(* PLC project v0.6.02_RefactorGateAndTest.project, CODESYS CODESYS V3.5 SP19 Patch 1 *)
(* stored: creationDateTime 2026-08-14T10:10:49.355835, modificationDateTime 2026-08-14T10:10:49.355835 *)

(* ═══════════════════════════════════════════════════════════════ 🛡️ ST_Safety_Emergency_Diag — Diagnostic et erreurs de la chaîne AU ─────────────────────────────────────────────────────────────── 📄 Produit par FB_Safety_EmergencyManagement (sortie Diag). Consommé par PRG_SUPERVISION_CFC et GVL_Troubleshooting. 🎯 Champs lecture seule — producteur unique = FB composite. ═══════════════════════════════════════════════════════════════ 📄 Docs : DOC/AF/AF_Partie-01_Analyse_Fonctionnelle_v2.0.md §8.2 DOC/AF/AF_Partie-03_Contrats_Composants_v2.1.md *)
TYPE ST_Safety_Emergency_Diag : STRUCT
  Error : BOOL;  (* 🔴 Synthèse : (ErrorId <> 0) *)
  ErrorId : WORD;  (* ❌ bit0 = RedundancyTestFailed (auto-test A/B), bit1 = EmergencyArmingFailed (timeout confirm contacteur) *)
  RedundancyTestFailed : BOOL;  (* 🔴 Canal A ou B resté collé/shunté détecté à l'auto-test — Reset requis (cause disparue) *)
  ArmFailed : BOOL;  (* 🔴 Impulsion envoyée mais contacteur puissance non confirmé sous 2 s — Reset + contacteur engagé requis *)
  LockoutActive : BOOL;  (* ⏳ Verrouillage temporel de 5 s entre tentatives de réarmement échouées *)
END_STRUCT;
END_TYPE

(* ═══════════════════════════════════════════════════════════════ ⚙️ ST_Safety_Emergency_InternalCmd — Structure de commande interne ─────────────────────────────────────────────────────────────── 📄 Transporte les ordres logiques entre le bloc de décision et le bloc de sortie de la boucle d'urgence. 🔒 Polarité maintien : TRUE = voie maintenue saine, FALSE = coupure demandée (conforme règle C1 — polarité explicite). ═══════════════════════════════════════════════════════════════ 📄 Docs : DOC/AF/AF_Partie-01_Analyse_Fonctionnelle_v2.0.md *)
TYPE ST_Safety_Emergency_InternalCmd : STRUCT
  MaintainA_Cmd : BOOL;  (* Ordre maintien canal A (TRUE = voie maintenue, FALSE = coupure demandée) *)
  MaintainB_Cmd : BOOL;  (* Ordre maintien canal B (TRUE = voie maintenue, FALSE = coupure demandée) *)
  ArmPulse_Cmd : BOOL;  (* Ordre impulsion de réarmement (TRUE = bobine réarmement activée) *)
END_STRUCT;
END_TYPE

(* ═══════════════════════════════════════════════════════════════ 🚦 ST_Safety_Emergency_State — État public de la chaîne d'arrêt d'urgence ─────────────────────────────────────────────────────────────── 📄 Produit par FB_Safety_EmergencyManagement (sortie State). Consommé par PRG_SUPERVISION_CFC → GVL_IHM.Modes.State pour IHM, et par GVL_Troubleshooting pour diagnostic. 🎯 Champs lecture seule — aucun lecteur n'est autorisé à l'écrire. ═══════════════════════════════════════════════════════════════ 📄 Docs : DOC/AF/AF_Partie-01_Analyse_Fonctionnelle_v2.0.md §8.2 DOC/AF/AF_Partie-03_Contrats_Composants_v2.1.md *)
TYPE ST_Safety_Emergency_State : STRUCT
  ChainOk : BOOL;  (* 🔗 Boucle AU fermée (EmergencyChainClosed_DI = TRUE) *)
  ContactorOk : BOOL;  (* 🔌 Contacteur puissance confirmé engagé (PowerContactorEngaged_DI = TRUE) *)
  Step : INT;  (* 🔢 Étape séquence armement : 0=IDLE, 1=TestA, 2=RestoreA, 3=TestB, 4=RestoreB, 5=Pulse, 6=Confirm *)
  Armable : BOOL;  (* 🟢 Réarmement possible maintenant : chain OK, step=0, pas de lockout, pas de redondance échouée, pas de contacteur déjà engagé *)
  ArmingBusy : BOOL;  (* ⏳ Séquence armement OU lockout en cours (nouvelle demande ignorée) *)
END_STRUCT;
END_TYPE

(* ═══════════════════════════════════════════════════════════════ 🔒 FB_Safety_EmergencyManagementOutput — Projection Physique Fail-Safe ─────────────────────────────────────────────────────────────── 🎯 Rôle : Enable gate + copie consignes logiques vers sorties physiques 🔒 Polarité : MaintainA/B_RQ en maintien (TRUE = voie saine) 📄 Docs : DOC/AF/AF_Partie-01_Analyse_Fonctionnelle/FB_Safety_EmergencyManagement_v1.1.md DOC/AF/AF_Partie-01_Analyse_Fonctionnelle_v2.0.md DOC/AF/AF_Partie-03_Contrats_Composants_v2.1.md *)
FUNCTION_BLOCK FB_Safety_EmergencyManagementOutput
  VAR_INPUT
    Enable : BOOL;  (* Active le pilote (FALSE = toutes sorties à FALSE) *)
    Cmd : ST_Safety_Emergency_InternalCmd;  (* Ordres logiques reçus du bloc logique *)
    ChainOk : BOOL;  (* Miroir EmergencyChainClosed (pour bus State) *)
    ContactorOk : BOOL;  (* Miroir PowerContactorEngaged (pour bus State) *)
    ArmingStep : INT;  (* Miroir ArmingSeqStep (pour bus State) *)
    Armable : BOOL;  (* Calculé par Logic (pour bus State) *)
    ArmingBusy : BOOL;  (* Calculé par Logic (pour bus State) *)
    Error : BOOL;  (* Miroir Error (pour bus Diag) *)
    ErrorId : WORD;  (* Miroir ErrorId (pour bus Diag) *)
    RedundancyTestFailed : BOOL;  (* Miroir (pour bus Diag) *)
    ArmFailed : BOOL;  (* Miroir (pour bus Diag) *)
    LockoutActive : BOOL;  (* Miroir (pour bus Diag) *)
  END_VAR
  VAR_OUTPUT
    MaintainA_RQ : BOOL;  (* ⚡ Sorties physiques terminales Vers relais maintien canal A — TRUE = voie maintenue, FALSE = coupure *)
    MaintainB_RQ : BOOL;  (* Vers relais maintien canal B — TRUE = voie maintenue, FALSE = coupure *)
    ArmPulse_RQ : BOOL;  (* Vers contacteur impulsion réarmement — TRUE = pulse actif *)
    State : ST_Safety_Emergency_State;  (* 🚦 Bus d'état public *)
    Diag : ST_Safety_Emergency_Diag;
  END_VAR

            

// === IMPLEMENTATION ===

IF NOT Enable THEN
    MaintainA_RQ   := FALSE;
    MaintainB_RQ   := FALSE;
    ArmPulse_RQ    := FALSE;

    State.ChainOk        := FALSE;
    State.ContactorOk    := FALSE;
    State.Step           := 0;
    State.Armable        := FALSE;
    State.ArmingBusy     := FALSE;

    Diag.Error                := FALSE;
    Diag.ErrorId              := 16#0000;
    Diag.RedundancyTestFailed := FALSE;
    Diag.ArmFailed            := FALSE;
    Diag.LockoutActive        := FALSE;
    RETURN;
END_IF;

// ⚡ Sorties physiques — écriture directe des ordres logiques
MaintainA_RQ := Cmd.MaintainA_Cmd;
MaintainB_RQ := Cmd.MaintainB_Cmd;
ArmPulse_RQ  := Cmd.ArmPulse_Cmd;

// 🚦 Bus d'état public
State.ChainOk        := ChainOk;
State.ContactorOk    := ContactorOk;
State.Step           := ArmingStep;
State.Armable        := Armable;
State.ArmingBusy     := ArmingBusy;

// 🛡️ Bus diagnostic public
Diag.Error                := Error;
Diag.ErrorId              := ErrorId;
Diag.RedundancyTestFailed := RedundancyTestFailed;
Diag.ArmFailed            := ArmFailed;
Diag.LockoutActive        := LockoutActive;

          
END_FUNCTION_BLOCK
